FUNCTION F_BaseplateChiller_Error : FB_BaseplateChiller
VAR_INPUT
END_VAR
VAR
	fbBaseplateChiller : FB_BaseplateChiller;
END_VAR

fbBaseplateChiller(bBaseplateChillerFlow := FALSE);
F_BaseplateChiller_Error := fbBaseplateChiller;

END_FUNCTION

(* stored: Version 1.1.0.1, ProductVersion 3.1.4020.14
   POU F_BaseplateChiller_Error: Id {1be9e493-d087-4dde-af8e-482905c4eb37}, SpecialFunc None *)
